FUNCTION_BLOCK FB_FL
VAR_INPUT
	Larm_in :BOOL;
	TID_in :INT;
END_VAR
VAR_OUTPUT
	Larm_ut :BOOL;
END_VAR
VAR
	TON_0: TON;
END_VAR

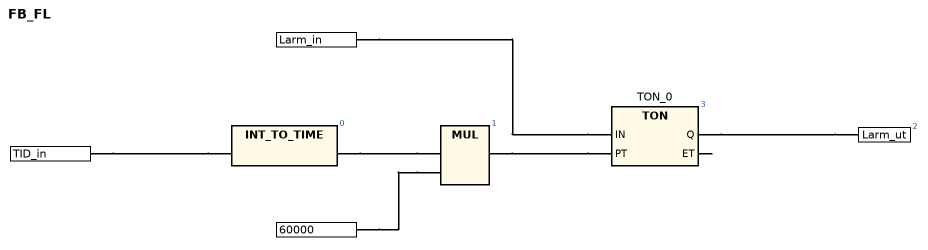
Larm_ut := TON_0.Q;
TON_0(IN := Larm_in, PT := INT_TO_TIME(TID_in) * 60000); // TON

END_FUNCTION_BLOCK

(* stored: Version 1.1.0.1, ProductVersion 3.1.4020.12
   POU FB_FL: Id {3e701fa6-6068-402f-ad1c-6072b011c5b2}, SpecialFunc None *)
